# EPICS autosave request: pgpEdtApp/Db/pgpEdt_settings.req
$(P)$(R)PixelSize
$(P)$(R)Baud
$(P)$(R)SSUS
$(P)$(R)Pack
$(P)$(R)VOut
$(P)$(R)SkipRow
$(P)$(R)SkipCol
$(P)$(R)FullNRow
$(P)$(R)FullNCol
$(P)$(R)CC
$(P)$(R)TrgPolarity
$(P)$(R)EvrPrescale
$(P)$(R)TrgCode
$(P)$(R)TrgDelay
$(P)$(R)TrgWidth
$(P)$(R)CmdInit
$(P)$(R)CmdFull
$(P)$(R)CmdROI
$(P)$(R)CmdEVR
$(P)$(R)CmdFree
$(P)$(R)CmdTPtn
$(P)$(R)ExposureMode
